{attribute addProperty BoxType "BK1120-0000-0017"}
{attribute addProperty Id "Term_377_KL1002KL1002_D229A9CA00"}
{attribute addProperty CRC "4081637326"}
{attribute addProperty SizeInBites "0"}
{attribute addProperty SizeInBytes "0"}
TYPE A_0004_BK1120_0000_0017_F348D7CE EXTENDS BK1120_4487A81F :
STRUCT
	{attribute addProperty Name "Term_377_KL1002"}
	Term_377_KL1002 : KL1002_D229A9CA;
END_STRUCT
END_TYPE

(* stored: Version 1.2.0.0, ProductVersion 3.1.4024.9
   DUT A_0004_BK1120_0000_0017_F348D7CE: Id {f3aee3c1-1701-486b-85eb-fdc6127ba039} *)
